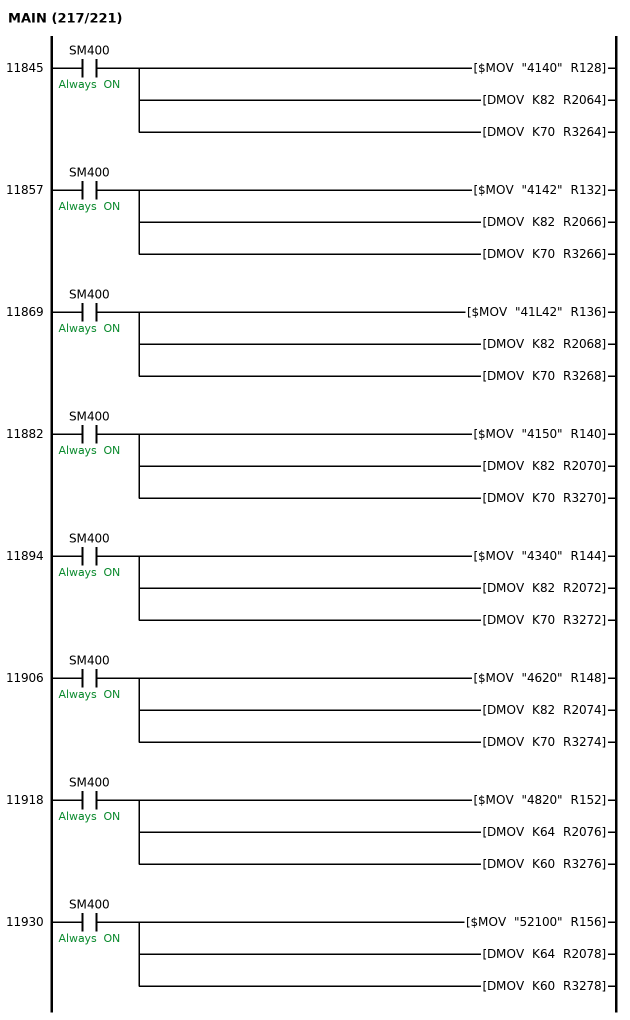
[picture p216: ladder of MAIN, rungs at steps 11845 to 11930]
11845 LD      SM400  ; Always  ON
      $MOV    "4140" R128
      DMOV    K82 R2064
      DMOV    K70 R3264
11857 LD      SM400  ; Always  ON
      $MOV    "4142" R132
      DMOV    K82 R2066
      DMOV    K70 R3266
11869 LD      SM400  ; Always  ON
      $MOV    "41L42" R136
      DMOV    K82 R2068
      DMOV    K70 R3268
11882 LD      SM400  ; Always  ON
      $MOV    "4150" R140
      DMOV    K82 R2070
      DMOV    K70 R3270
11894 LD      SM400  ; Always  ON
      $MOV    "4340" R144
      DMOV    K82 R2072
      DMOV    K70 R3272
11906 LD      SM400  ; Always  ON
      $MOV    "4620" R148
      DMOV    K82 R2074
      DMOV    K70 R3274
11918 LD      SM400  ; Always  ON
      $MOV    "4820" R152
      DMOV    K64 R2076
      DMOV    K60 R3276
11930 LD      SM400  ; Always  ON
      $MOV    "52100" R156
      DMOV    K64 R2078
      DMOV    K60 R3278
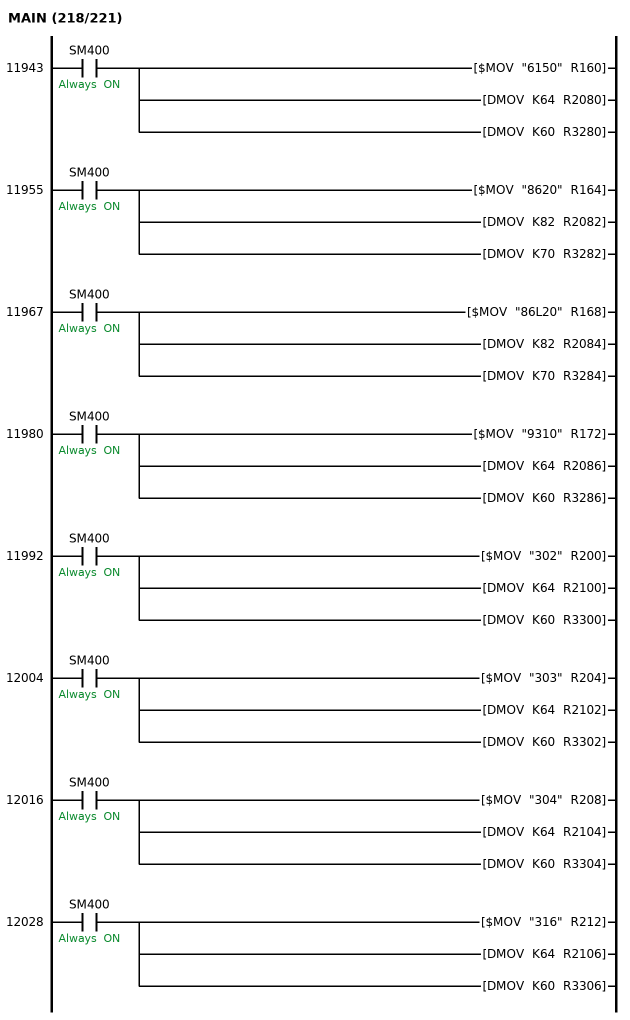
11943 LD      SM400  ; Always  ON
      $MOV    "6150" R160
      DMOV    K64 R2080
      DMOV    K60 R3280
11955 LD      SM400  ; Always  ON
      $MOV    "8620" R164
      DMOV    K82 R2082
      DMOV    K70 R3282
11967 LD      SM400  ; Always  ON
      $MOV    "86L20" R168
      DMOV    K82 R2084
      DMOV    K70 R3284
11980 LD      SM400  ; Always  ON
      $MOV    "9310" R172
      DMOV    K64 R2086
      DMOV    K60 R3286
11992 LD      SM400  ; Always  ON
      $MOV    "302" R200
      DMOV    K64 R2100
      DMOV    K60 R3300
12004 LD      SM400  ; Always  ON
      $MOV    "303" R204
      DMOV    K64 R2102
      DMOV    K60 R3302
12016 LD      SM400  ; Always  ON
      $MOV    "304" R208
      DMOV    K64 R2104
      DMOV    K60 R3304
12028 LD      SM400  ; Always  ON
      $MOV    "316" R212
      DMOV    K64 R2106
      DMOV    K60 R3306
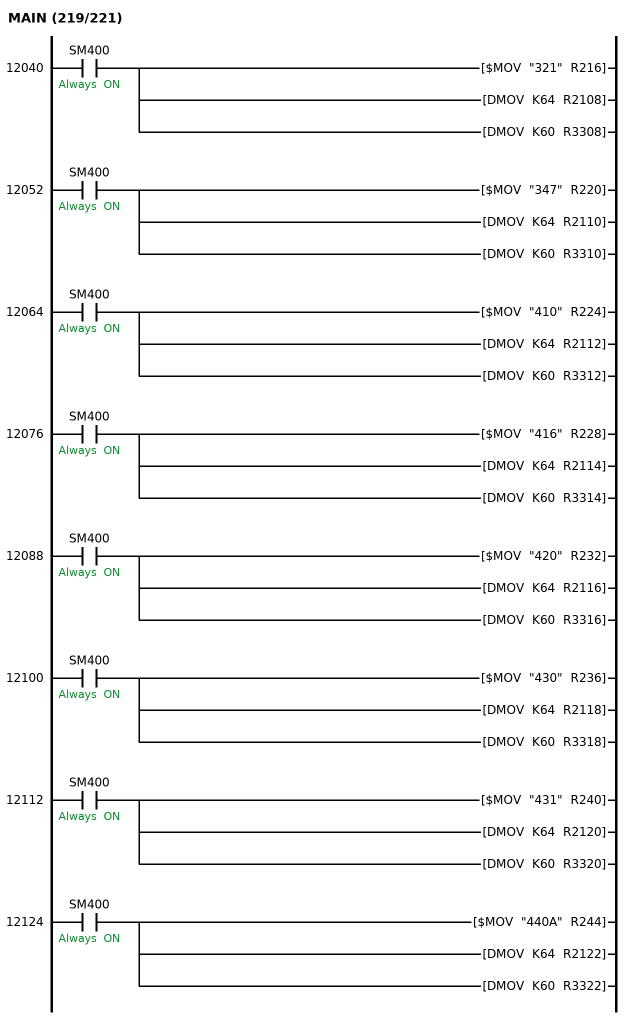
12040 LD      SM400  ; Always  ON
      $MOV    "321" R216
      DMOV    K64 R2108
      DMOV    K60 R3308
12052 LD      SM400  ; Always  ON
      $MOV    "347" R220
      DMOV    K64 R2110
      DMOV    K60 R3310
12064 LD      SM400  ; Always  ON
      $MOV    "410" R224
      DMOV    K64 R2112
      DMOV    K60 R3312
12076 LD      SM400  ; Always  ON
      $MOV    "416" R228
      DMOV    K64 R2114
      DMOV    K60 R3314
12088 LD      SM400  ; Always  ON
      $MOV    "420" R232
      DMOV    K64 R2116
      DMOV    K60 R3316
12100 LD      SM400  ; Always  ON
      $MOV    "430" R236
      DMOV    K64 R2118
      DMOV    K60 R3318
12112 LD      SM400  ; Always  ON
      $MOV    "431" R240
      DMOV    K64 R2120
      DMOV    K60 R3320
12124 LD      SM400  ; Always  ON
      $MOV    "440A" R244
      DMOV    K64 R2122
      DMOV    K60 R3322
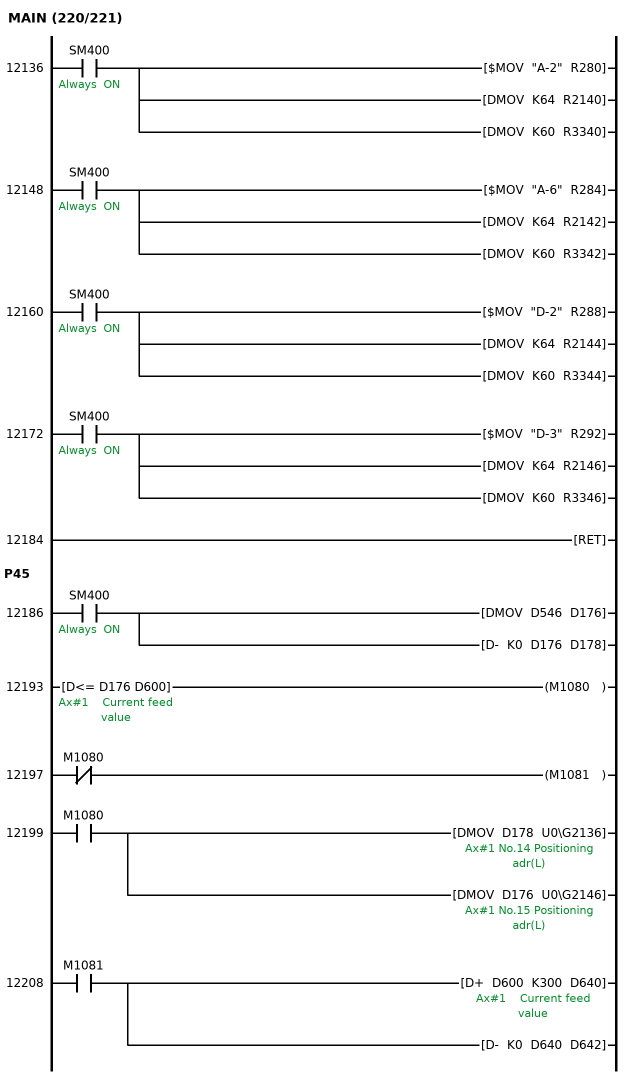
12136 LD      SM400  ; Always  ON
      $MOV    "A-2" R280
      DMOV    K64 R2140
      DMOV    K60 R3340
12148 LD      SM400  ; Always  ON
      $MOV    "A-6" R284
      DMOV    K64 R2142
      DMOV    K60 R3342
12160 LD      SM400  ; Always  ON
      $MOV    "D-2" R288
      DMOV    K64 R2144
      DMOV    K60 R3344
12172 LD      SM400  ; Always  ON
      $MOV    "D-3" R292
      DMOV    K64 R2146
      DMOV    K60 R3346
12184 RET
      P45
12186 LD      SM400  ; Always  ON
      DMOV    D546 D176
      D-      K0 D176 D178
12193 LDD<=   D176 D600  ; Ax#1    Current feed    value
      OUT     M1080
12197 LDI     M1080
      OUT     M1081
12199 LD      M1080
      DMOV    D178 U0\G2136  ; Ax#1 No.14 Positioning adr(L)
      DMOV    D176 U0\G2146  ; Ax#1 No.15 Positioning adr(L)
12208 LD      M1081
      D+      D600 K300 D640
      D-      K0 D640 D642
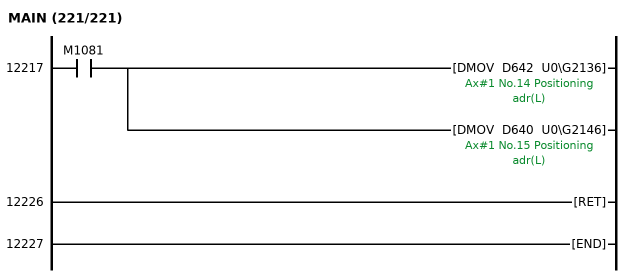
12217 LD      M1081
      DMOV    D642 U0\G2136
      DMOV    D640 U0\G2146
12226 RET
12227 END
END_PROGRAM

PROGRAM HMS
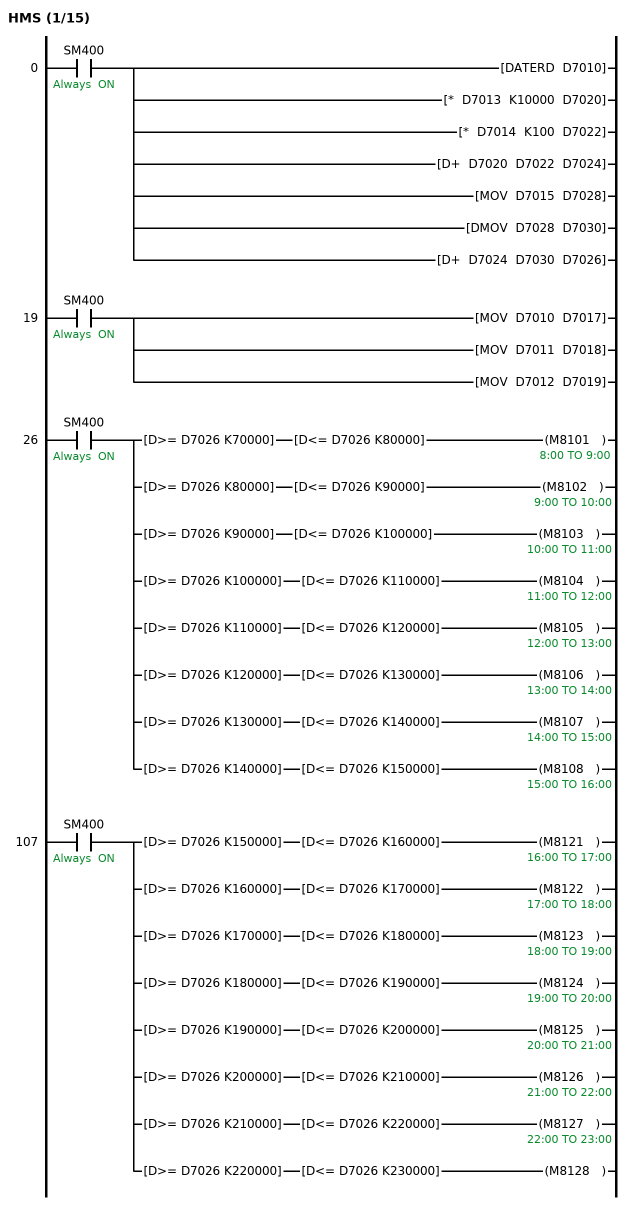
0     LD      SM400  ; Always  ON
      DATERD  D7010
      *       D7013 K10000 D7020
      *       D7014 K100 D7022
      D+      D7020 D7022 D7024
      MOV     D7015 D7028
      DMOV    D7028 D7030
      D+      D7024 D7030 D7026
19    LD      SM400  ; Always  ON
      MOV     D7010 D7017
      MOV     D7011 D7018
      MOV     D7012 D7019
26    LD      SM400  ; Always  ON
      MPS
      ANDD>=  D7026 K70000
      ANDD<=  D7026 K80000
      OUT     M8101  ; 8:00 TO 9:00
      MRD
      ANDD>=  D7026 K80000
      ANDD<=  D7026 K90000
      OUT     M8102  ; 9:00 TO 10:00
      MRD
      ANDD>=  D7026 K90000
      ANDD<=  D7026 K100000
      OUT     M8103  ; 10:00 TO 11:00
      MRD
      ANDD>=  D7026 K100000
      ANDD<=  D7026 K110000
      OUT     M8104  ; 11:00 TO 12:00
      MRD
      ANDD>=  D7026 K110000
      ANDD<=  D7026 K120000
      OUT     M8105  ; 12:00 TO 13:00
      MRD
      ANDD>=  D7026 K120000
      ANDD<=  D7026 K130000
      OUT     M8106  ; 13:00 TO 14:00
      MRD
      ANDD>=  D7026 K130000
      ANDD<=  D7026 K140000
      OUT     M8107  ; 14:00 TO 15:00
      MPP
      ANDD>=  D7026 K140000
      ANDD<=  D7026 K150000
      OUT     M8108  ; 15:00 TO 16:00
107   LD      SM400  ; Always  ON
      MPS
      ANDD>=  D7026 K150000
      ANDD<=  D7026 K160000
      OUT     M8121  ; 16:00 TO 17:00
      MRD
      ANDD>=  D7026 K160000
      ANDD<=  D7026 K170000
      OUT     M8122  ; 17:00 TO 18:00
      MRD
      ANDD>=  D7026 K170000
      ANDD<=  D7026 K180000
      OUT     M8123  ; 18:00 TO 19:00
      MRD
      ANDD>=  D7026 K180000
      ANDD<=  D7026 K190000
      OUT     M8124  ; 19:00 TO 20:00
      MRD
      ANDD>=  D7026 K190000
      ANDD<=  D7026 K200000
      OUT     M8125  ; 20:00 TO 21:00
      MRD
      ANDD>=  D7026 K200000
      ANDD<=  D7026 K210000
      OUT     M8126  ; 21:00 TO 22:00
      MRD
      ANDD>=  D7026 K210000
      ANDD<=  D7026 K220000
      OUT     M8127  ; 22:00 TO 23:00
      MPP
      ANDD>=  D7026 K220000
      ANDD<=  D7026 K230000
      OUT     M8128
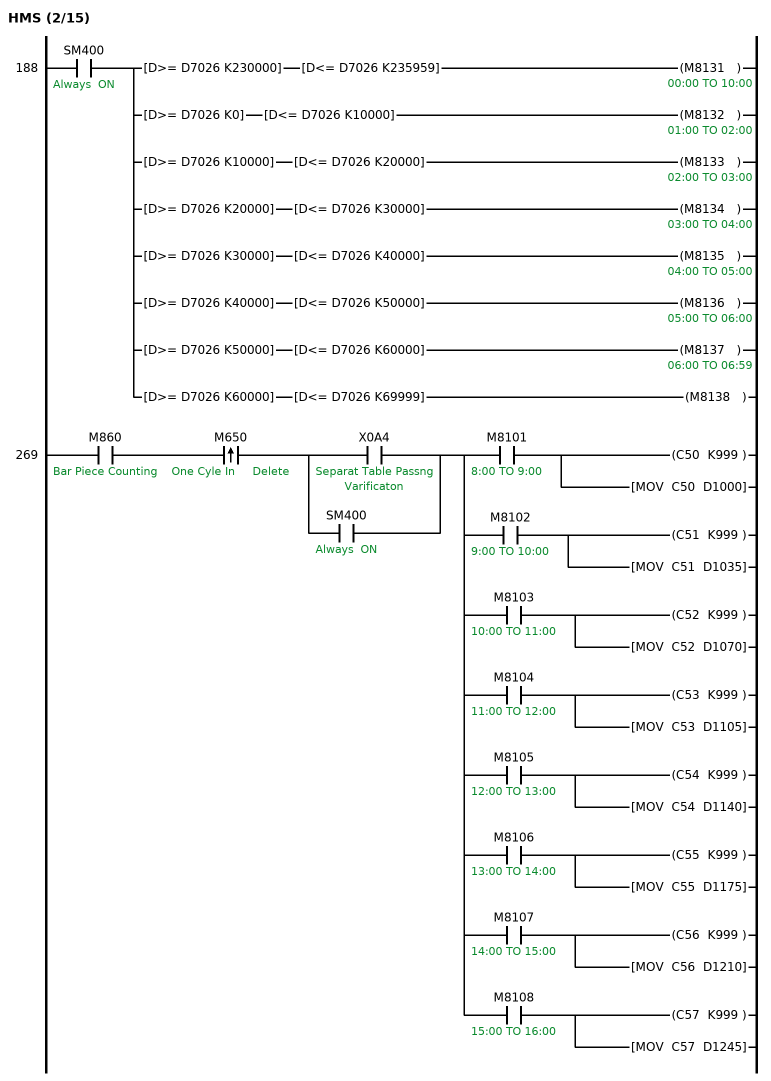
188   LD      SM400  ; Always  ON
      MPS
      ANDD>=  D7026 K230000
      ANDD<=  D7026 K235959
      OUT     M8131  ; 00:00 TO 10:00
      MRD
      ANDD>=  D7026 K0
      ANDD<=  D7026 K10000
      OUT     M8132  ; 01:00 TO 02:00
      MRD
      ANDD>=  D7026 K10000
      ANDD<=  D7026 K20000
      OUT     M8133  ; 02:00 TO 03:00
      MRD
      ANDD>=  D7026 K20000
      ANDD<=  D7026 K30000
      OUT     M8134  ; 03:00 TO 04:00
      MRD
      ANDD>=  D7026 K30000
      ANDD<=  D7026 K40000
      OUT     M8135  ; 04:00 TO 05:00
      MRD
      ANDD>=  D7026 K40000
      ANDD<=  D7026 K50000
      OUT     M8136  ; 05:00 TO 06:00
      MRD
      ANDD>=  D7026 K50000
      ANDD<=  D7026 K60000
      OUT     M8137  ; 06:00 TO 06:59
      MPP
      ANDD>=  D7026 K60000
      ANDD<=  D7026 K69999
      OUT     M8138
269   LD      M860  ; Bar Piece Counting
      ANDP    M650  ; One Cyle In     Delete
      LD      X0A4  ; Separat Table Passng Varificaton
      OR      SM400  ; Always  ON
      ANB
      MPS
      AND     M8101  ; 8:00 TO 9:00
      OUT     C50 K999
      MOV     C50 D1000
      MRD
      AND     M8102  ; 9:00 TO 10:00
      OUT     C51 K999
      MOV     C51 D1035
      MRD
      AND     M8103  ; 10:00 TO 11:00
      OUT     C52 K999
      MOV     C52 D1070
      MRD
      AND     M8104  ; 11:00 TO 12:00
      OUT     C53 K999
      MOV     C53 D1105
      MRD
      AND     M8105  ; 12:00 TO 13:00
      OUT     C54 K999
      MOV     C54 D1140
      MRD
      AND     M8106  ; 13:00 TO 14:00
      OUT     C55 K999
      MOV     C55 D1175
      MRD
      AND     M8107  ; 14:00 TO 15:00
      OUT     C56 K999
      MOV     C56 D1210
      MPP
      AND     M8108  ; 15:00 TO 16:00
      OUT     C57 K999
      MOV     C57 D1245
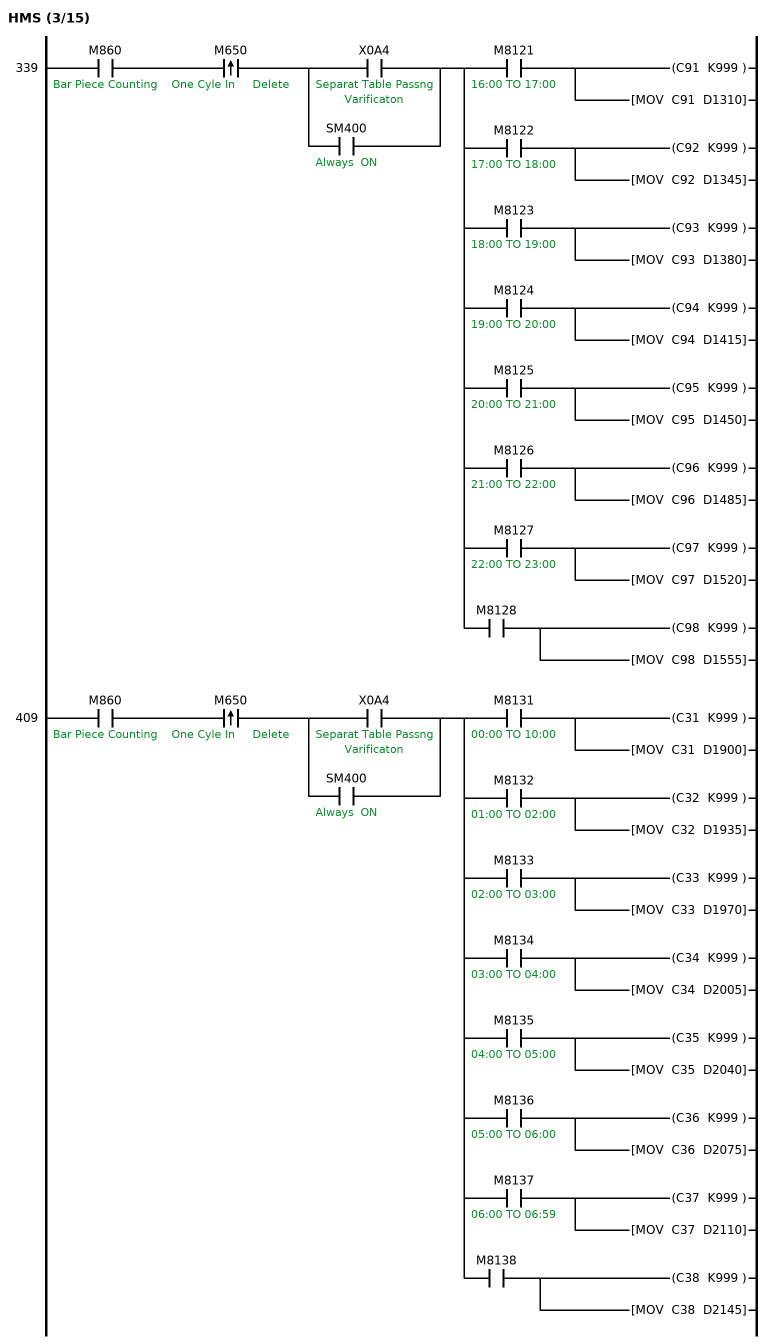
339   LD      M860  ; Bar Piece Counting
      ANDP    M650  ; One Cyle In     Delete
      LD      X0A4  ; Separat Table Passng Varificaton
      OR      SM400  ; Always  ON
      ANB
      MPS
      AND     M8121  ; 16:00 TO 17:00
      OUT     C91 K999
      MOV     C91 D1310
      MRD
      AND     M8122  ; 17:00 TO 18:00
      OUT     C92 K999
      MOV     C92 D1345
      MRD
      AND     M8123  ; 18:00 TO 19:00
      OUT     C93 K999
      MOV     C93 D1380
      MRD
      AND     M8124  ; 19:00 TO 20:00
      OUT     C94 K999
      MOV     C94 D1415
      MRD
      AND     M8125  ; 20:00 TO 21:00
      OUT     C95 K999
      MOV     C95 D1450
      MRD
      AND     M8126  ; 21:00 TO 22:00
      OUT     C96 K999
      MOV     C96 D1485
      MRD
      AND     M8127  ; 22:00 TO 23:00
      OUT     C97 K999
      MOV     C97 D1520
      MPP
      AND     M8128
      OUT     C98 K999
      MOV     C98 D1555
409   LD      M860  ; Bar Piece Counting
      ANDP    M650  ; One Cyle In     Delete
      LD      X0A4  ; Separat Table Passng Varificaton
      OR      SM400  ; Always  ON
      ANB
      MPS
      AND     M8131  ; 00:00 TO 10:00
      OUT     C31 K999
      MOV     C31 D1900
      MRD
      AND     M8132  ; 01:00 TO 02:00
      OUT     C32 K999
      MOV     C32 D1935
      MRD
      AND     M8133  ; 02:00 TO 03:00
      OUT     C33 K999
      MOV     C33 D1970
      MRD
      AND     M8134  ; 03:00 TO 04:00
      OUT     C34 K999
      MOV     C34 D2005
      MRD
      AND     M8135  ; 04:00 TO 05:00
      OUT     C35 K999
      MOV     C35 D2040
      MRD
      AND     M8136  ; 05:00 TO 06:00
      OUT     C36 K999
      MOV     C36 D2075
      MRD
      AND     M8137  ; 06:00 TO 06:59
      OUT     C37 K999
      MOV     C37 D2110
      MPP
      AND     M8138
      OUT     C38 K999
      MOV     C38 D2145
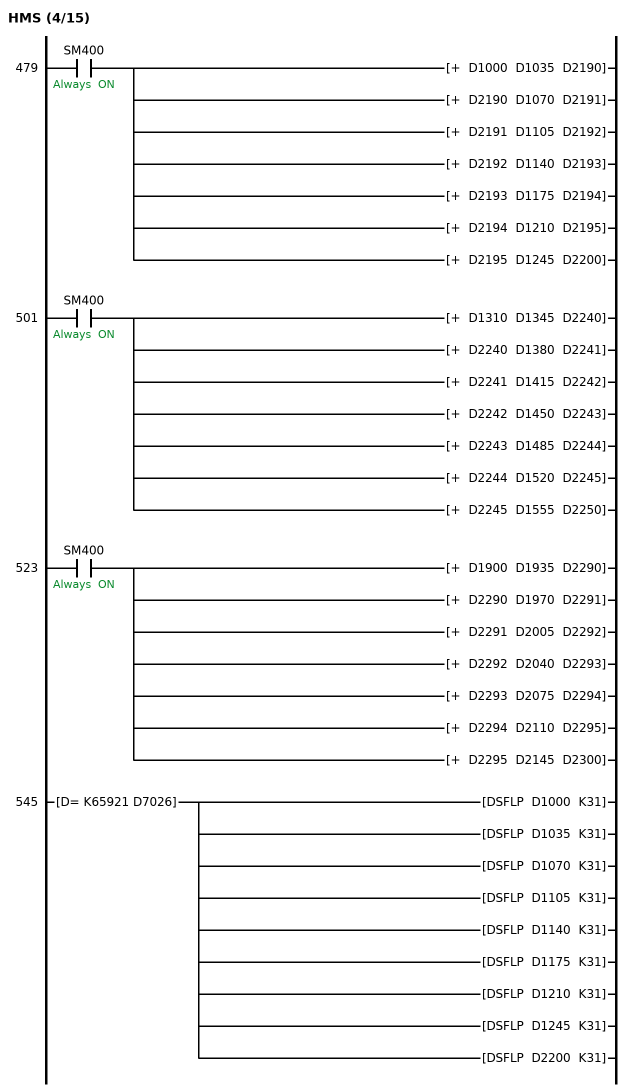
479   LD      SM400  ; Always  ON
      +       D1000 D1035 D2190
      +       D2190 D1070 D2191
      +       D2191 D1105 D2192
      +       D2192 D1140 D2193
      +       D2193 D1175 D2194
      +       D2194 D1210 D2195
      +       D2195 D1245 D2200
501   LD      SM400  ; Always  ON
      +       D1310 D1345 D2240
      +       D2240 D1380 D2241
      +       D2241 D1415 D2242
      +       D2242 D1450 D2243
      +       D2243 D1485 D2244
      +       D2244 D1520 D2245
      +       D2245 D1555 D2250
523   LD      SM400  ; Always  ON
      +       D1900 D1935 D2290
      +       D2290 D1970 D2291
      +       D2291 D2005 D2292
      +       D2292 D2040 D2293
      +       D2293 D2075 D2294
      +       D2294 D2110 D2295
      +       D2295 D2145 D2300
545   LDD=    K65921 D7026
      DSFLP   D1000 K31
      DSFLP   D1035 K31
      DSFLP   D1070 K31
      DSFLP   D1105 K31
      DSFLP   D1140 K31
      DSFLP   D1175 K31
      DSFLP   D1210 K31
      DSFLP   D1245 K31
      DSFLP   D2200 K31
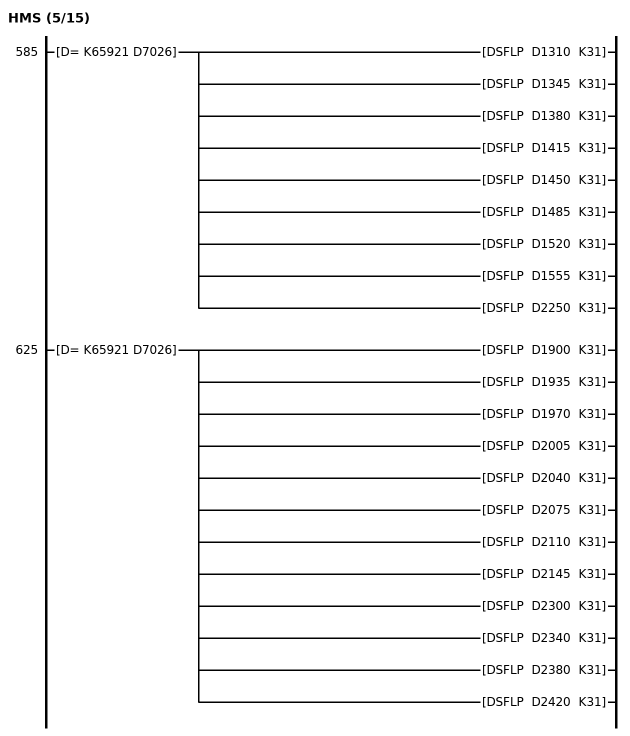
585   LDD=    K65921 D7026
      DSFLP   D1310 K31
      DSFLP   D1345 K31
      DSFLP   D1380 K31
      DSFLP   D1415 K31
      DSFLP   D1450 K31
      DSFLP   D1485 K31
      DSFLP   D1520 K31
      DSFLP   D1555 K31
      DSFLP   D2250 K31
625   LDD=    K65921 D7026
      DSFLP   D1900 K31
      DSFLP   D1935 K31
      DSFLP   D1970 K31
      DSFLP   D2005 K31
      DSFLP   D2040 K31
      DSFLP   D2075 K31
      DSFLP   D2110 K31
      DSFLP   D2145 K31
      DSFLP   D2300 K31
      DSFLP   D2340 K31
      DSFLP   D2380 K31
      DSFLP   D2420 K31
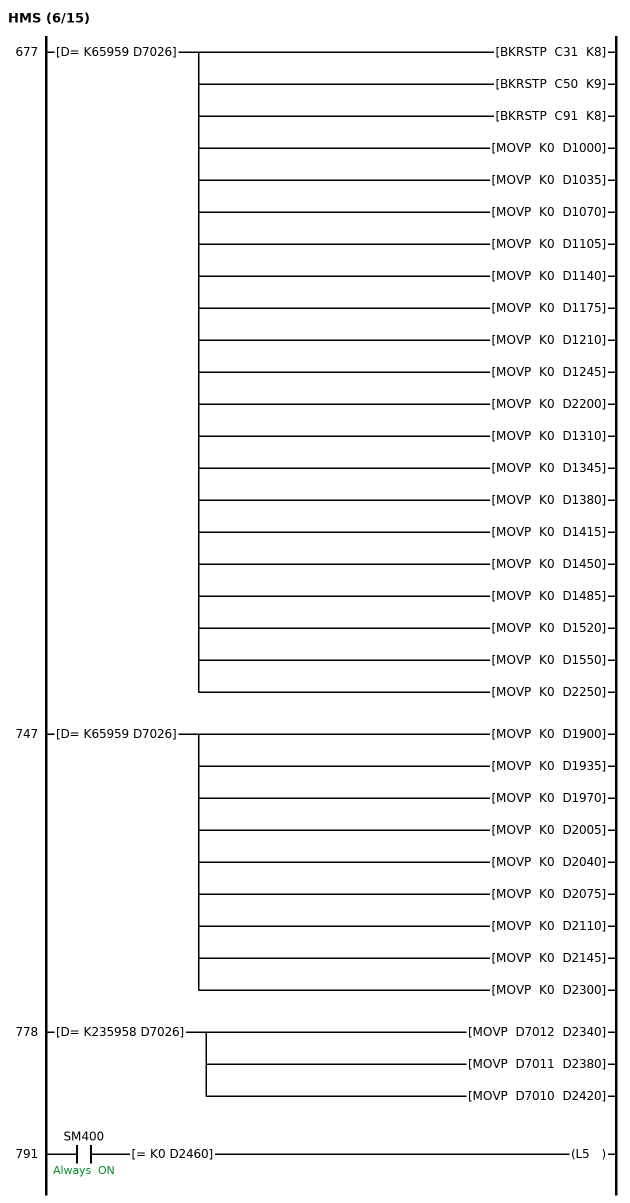
677   LDD=    K65959 D7026
      BKRSTP  C31 K8
      BKRSTP  C50 K9
      BKRSTP  C91 K8
      MOVP    K0 D1000
      MOVP    K0 D1035
      MOVP    K0 D1070
      MOVP    K0 D1105
      MOVP    K0 D1140
      MOVP    K0 D1175
      MOVP    K0 D1210
      MOVP    K0 D1245
      MOVP    K0 D2200
      MOVP    K0 D1310
      MOVP    K0 D1345
      MOVP    K0 D1380
      MOVP    K0 D1415
      MOVP    K0 D1450
      MOVP    K0 D1485
      MOVP    K0 D1520
      MOVP    K0 D1550
      MOVP    K0 D2250
747   LDD=    K65959 D7026
      MOVP    K0 D1900
      MOVP    K0 D1935
      MOVP    K0 D1970
      MOVP    K0 D2005
      MOVP    K0 D2040
      MOVP    K0 D2075
      MOVP    K0 D2110
      MOVP    K0 D2145
      MOVP    K0 D2300
778   LDD=    K235958 D7026
      MOVP    D7012 D2340
      MOVP    D7011 D2380
      MOVP    D7010 D2420
791   LD      SM400  ; Always  ON
      AND=    K0 D2460
      OUT     L5
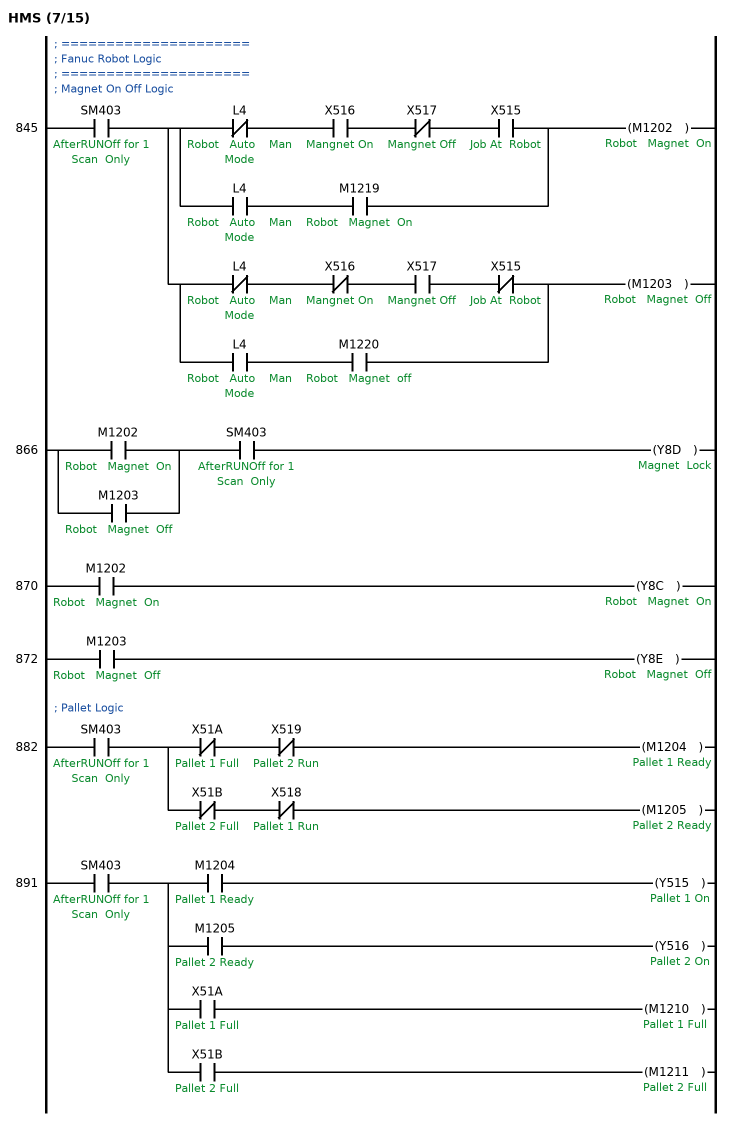
; =====================
; Fanuc Robot Logic
; =====================
; Magnet On Off Logic
845   LD      SM403  ; AfterRUNOff for 1 Scan  Only
      MPS
      LDI     L4  ; Robot   Auto    Man     Mode
      AND     X516  ; Mangnet On
      ANI     X517  ; Mangnet Off
      AND     X515  ; Job At  Robot
      LD      L4  ; Robot   Auto    Man     Mode
      AND     M1219  ; Robot   Magnet  On
      ORB
      ANB
      OUT     M1202  ; Robot   Magnet  On
      MPP
      LDI     L4  ; Robot   Auto    Man     Mode
      ANI     X516  ; Mangnet On
      AND     X517  ; Mangnet Off
      ANI     X515  ; Job At  Robot
      LD      L4  ; Robot   Auto    Man     Mode
      AND     M1220  ; Robot   Magnet  off
      ORB
      ANB
      OUT     M1203  ; Robot   Magnet  Off
866   LD      M1202  ; Robot   Magnet  On
      OR      M1203  ; Robot   Magnet  Off
      AND     SM403  ; AfterRUNOff for 1 Scan  Only
      OUT     Y8D  ; Magnet  Lock
870   LD      M1202  ; Robot   Magnet  On
      OUT     Y8C  ; Robot   Magnet  On
872   LD      M1203  ; Robot   Magnet  Off
      OUT     Y8E  ; Robot   Magnet  Off
; Pallet Logic
882   LD      SM403  ; AfterRUNOff for 1 Scan  Only
      MPS
      ANI     X51A  ; Pallet 1 Full
      ANI     X519  ; Pallet 2 Run
      OUT     M1204  ; Pallet 1 Ready
      MPP
      ANI     X51B  ; Pallet 2 Full
      ANI     X518  ; Pallet 1 Run
      OUT     M1205  ; Pallet 2 Ready
891   LD      SM403  ; AfterRUNOff for 1 Scan  Only
      MPS
      AND     M1204  ; Pallet 1 Ready
      OUT     Y515  ; Pallet 1 On
      MRD
      AND     M1205  ; Pallet 2 Ready
      OUT     Y516  ; Pallet 2 On
      MRD
      AND     X51A  ; Pallet 1 Full
      OUT     M1210  ; Pallet 1 Full
      MPP
      AND     X51B  ; Pallet 2 Full
      OUT     M1211  ; Pallet 2 Full
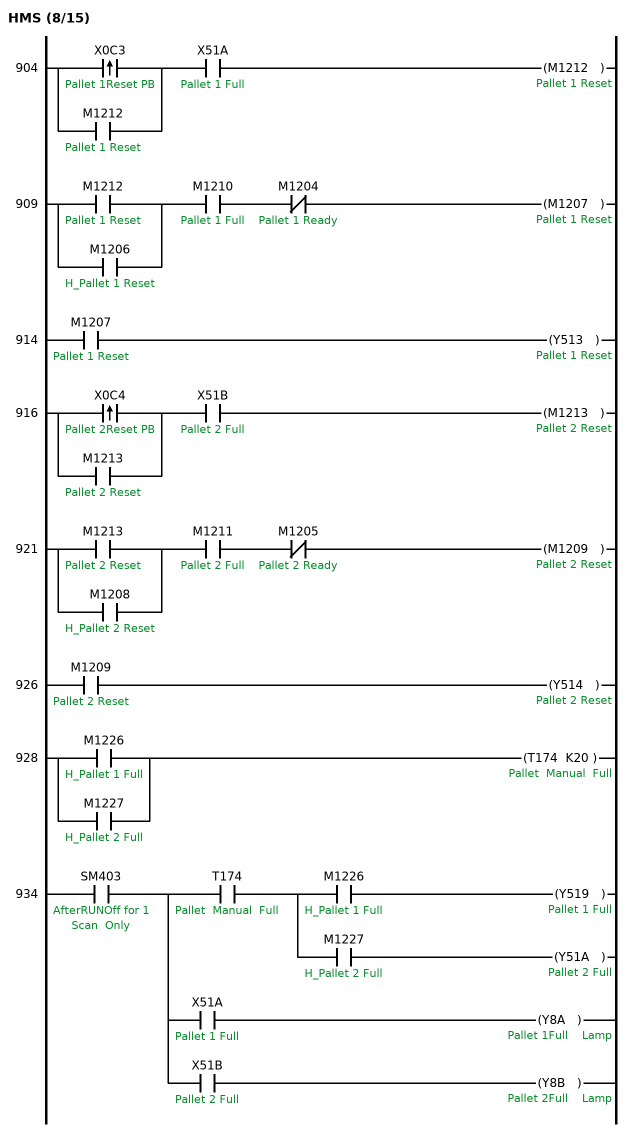
904   LDP     X0C3  ; Pallet 1Reset PB
      OR      M1212  ; Pallet 1 Reset
      AND     X51A  ; Pallet 1 Full
      OUT     M1212  ; Pallet 1 Reset
909   LD      M1212  ; Pallet 1 Reset
      OR      M1206  ; H_Pallet 1 Reset
      AND     M1210  ; Pallet 1 Full
      ANI     M1204  ; Pallet 1 Ready
      OUT     M1207  ; Pallet 1 Reset
914   LD      M1207  ; Pallet 1 Reset
      OUT     Y513  ; Pallet 1 Reset
916   LDP     X0C4  ; Pallet 2Reset PB
      OR      M1213  ; Pallet 2 Reset
      AND     X51B  ; Pallet 2 Full
      OUT     M1213  ; Pallet 2 Reset
921   LD      M1213  ; Pallet 2 Reset
      OR      M1208  ; H_Pallet 2 Reset
      AND     M1211  ; Pallet 2 Full
      ANI     M1205  ; Pallet 2 Ready
      OUT     M1209  ; Pallet 2 Reset
926   LD      M1209  ; Pallet 2 Reset
      OUT     Y514  ; Pallet 2 Reset
928   LD      M1226  ; H_Pallet 1 Full
      OR      M1227  ; H_Pallet 2 Full
      OUT     T174 K20  ; Pallet  Manual  Full
934   LD      SM403  ; AfterRUNOff for 1 Scan  Only
      MPS
      AND     T174  ; Pallet  Manual  Full
      MPS
      AND     M1226  ; H_Pallet 1 Full
      OUT     Y519  ; Pallet 1 Full
      MPP
      AND     M1227  ; H_Pallet 2 Full
      OUT     Y51A  ; Pallet 2 Full
      MRD
      AND     X51A  ; Pallet 1 Full
      OUT     Y8A  ; Pallet 1Full    Lamp
      MPP
      AND     X51B  ; Pallet 2 Full
      OUT     Y8B  ; Pallet 2Full    Lamp
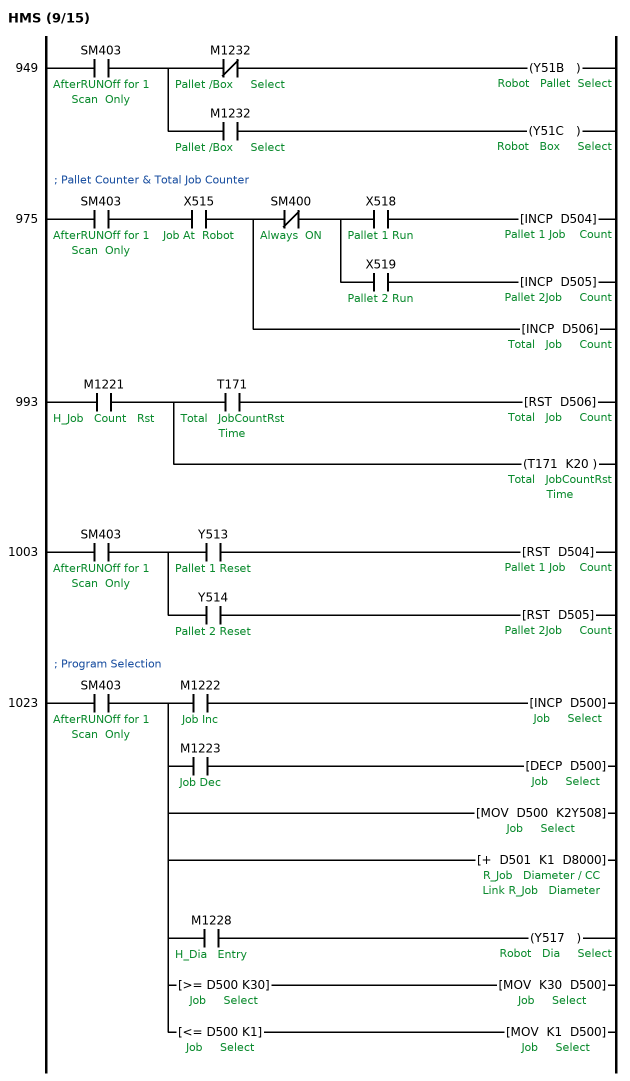
949   LD      SM403  ; AfterRUNOff for 1 Scan  Only
      MPS
      ANI     M1232  ; Pallet /Box     Select
      OUT     Y51B  ; Robot   Pallet  Select
      MPP
      AND     M1232  ; Pallet /Box     Select
      OUT     Y51C  ; Robot   Box     Select
; Pallet Counter & Total Job Counter
975   LD      SM403  ; AfterRUNOff for 1 Scan  Only
      AND     X515  ; Job At  Robot
      MPS
      ANI     SM400  ; Always  ON
      MPS
      AND     X518  ; Pallet 1 Run
      INCP    D504  ; Pallet 1 Job    Count
      MPP
      AND     X519  ; Pallet 2 Run
      INCP    D505  ; Pallet 2Job     Count
      MPP
      INCP    D506  ; Total   Job     Count
993   LD      M1221  ; H_Job   Count   Rst
      MPS
      AND     T171  ; Total   JobCountRst Time
      RST     D506  ; Total   Job     Count
      MPP
      OUT     T171 K20  ; Total   JobCountRst Time
1003  LD      SM403  ; AfterRUNOff for 1 Scan  Only
      MPS
      AND     Y513  ; Pallet 1 Reset
      RST     D504  ; Pallet 1 Job    Count
      MPP
      AND     Y514  ; Pallet 2 Reset
      RST     D505  ; Pallet 2Job     Count
; Program Selection
1023  LD      SM403  ; AfterRUNOff for 1 Scan  Only
      MPS
      AND     M1222  ; Job Inc
      INCP    D500  ; Job     Select
      MRD
      AND     M1223  ; Job Dec
      DECP    D500
      MPP
      MOV     D500 K2Y508  ; PNS 1   Style 1
      +       D501 K1 D8000  ; R_Job   Diameter / CC Link R_Job   Diameter
      MPS
      AND     M1228  ; H_Dia   Entry
      OUT     Y517  ; Robot   Dia     Select
      MRD
      AND>=   D500 K30  ; Job     Select
      MOV     K30 D500
      MPP
      AND<=   D500 K1  ; Job     Select
      MOV     K1 D500
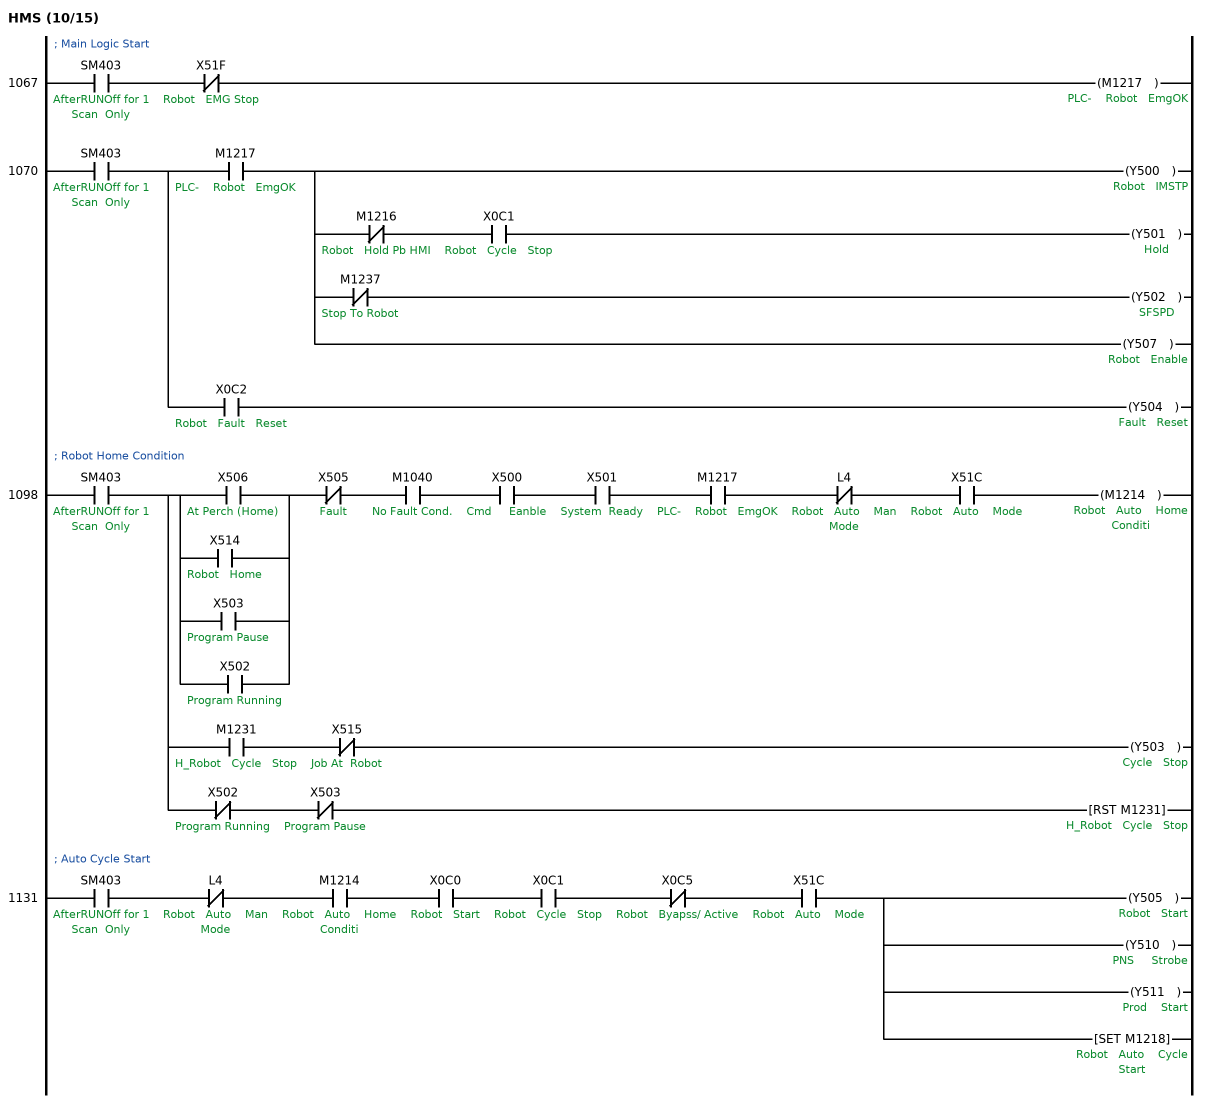
; Main Logic Start
1067  LD      SM403  ; AfterRUNOff for 1 Scan  Only
      ANI     X51F  ; Robot   EMG Stop
      OUT     M1217  ; PLC-    Robot   EmgOK
1070  LD      SM403  ; AfterRUNOff for 1 Scan  Only
      MPS
      AND     M1217  ; PLC-    Robot   EmgOK
      OUT     Y500  ; Robot   IMSTP
      MPS
      ANI     M1216  ; Robot   Hold Pb HMI
      AND     X0C1  ; Robot   Cycle   Stop
      OUT     Y501  ; Hold
      MRD
      ANI     M1237  ; Stop To Robot
      OUT     Y502  ; SFSPD
      MPP
      OUT     Y507  ; Robot   Enable
      MPP
      AND     X0C2  ; Robot   Fault   Reset
      OUT     Y504  ; Fault   Reset
; Robot Home Condition
1098  LD      SM403  ; AfterRUNOff for 1 Scan  Only
      MPS
      LD      X506  ; At Perch (Home)
      OR      X514  ; Robot   Home
      OR      X503  ; Program Pause
      OR      X502  ; Program Running
      ANB
      ANI     X505  ; Fault
      AND     M1040  ; No Fault Cond.
      AND     X500  ; Cmd     Eanble
      AND     X501  ; System  Ready
      AND     M1217  ; PLC-    Robot   EmgOK
      ANI     L4  ; Robot   Auto    Man     Mode
      AND     X51C  ; Robot   Auto    Mode
      OUT     M1214  ; Robot   Auto    Home    Conditi
      MRD
      AND     M1231  ; H_Robot   Cycle   Stop
      ANI     X515  ; Job At  Robot
      OUT     Y503  ; Cycle   Stop
      MPP
      ANI     X502  ; Program Running
      ANI     X503  ; Program Pause
      RST     M1231  ; H_Robot   Cycle   Stop
; Auto Cycle Start
1131  LD      SM403  ; AfterRUNOff for 1 Scan  Only
      ANI     L4  ; Robot   Auto    Man     Mode
      AND     M1214  ; Robot   Auto    Home    Conditi
      AND     X0C0  ; Robot   Start
      AND     X0C1  ; Robot   Cycle   Stop
      ANI     X0C5  ; Robot   Byapss/ Active
      AND     X51C  ; Robot   Auto    Mode
      OUT     Y505  ; Robot   Start
      OUT     Y510  ; PNS     Strobe
      OUT     Y511  ; Prod    Start
      SET     M1218  ; Robot   Auto    Cycle   Start
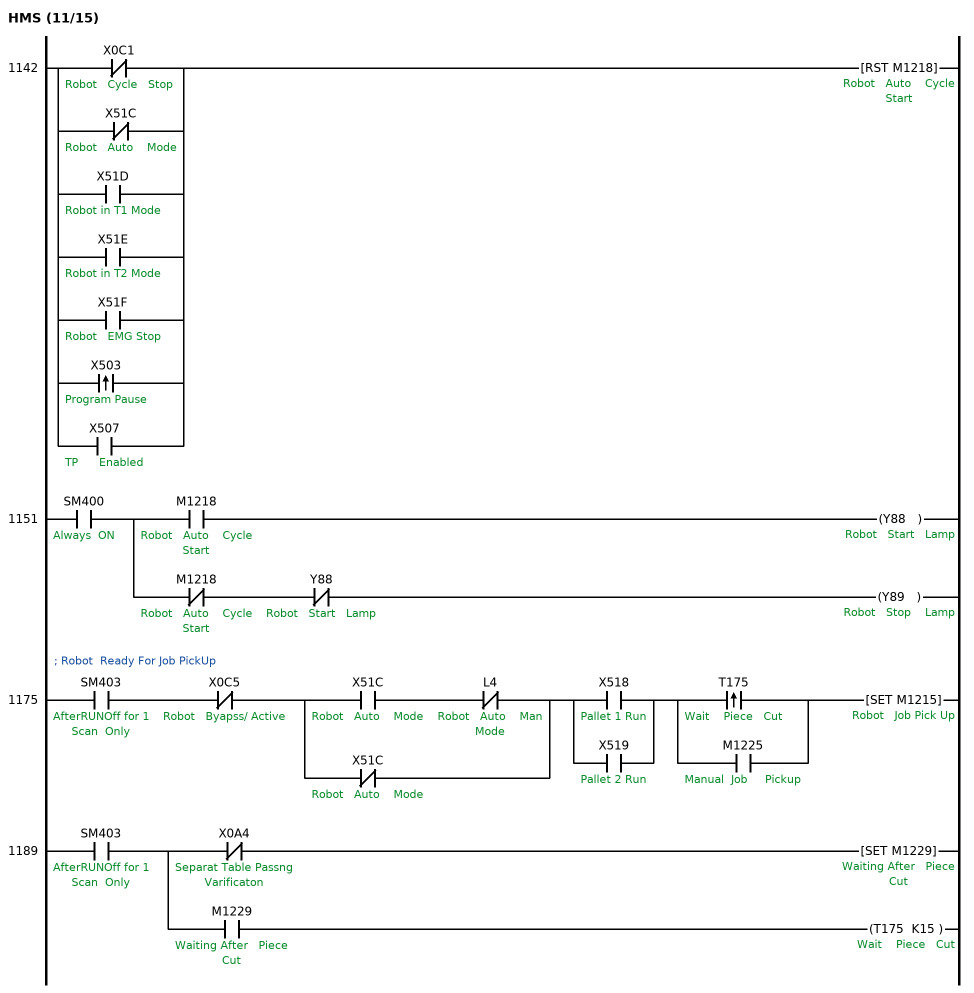
1142  LDI     X0C1  ; Robot   Cycle   Stop
      ORI     X51C  ; Robot   Auto    Mode
      OR      X51D  ; Robot in T1 Mode
      OR      X51E  ; Robot in T2 Mode
      OR      X51F  ; Robot   EMG Stop
      ORP     X503  ; Program Pause
      OR      X507  ; TP      Enabled
      RST     M1218  ; Robot   Auto    Cycle   Start
1151  LD      SM400  ; Always  ON
      MPS
      AND     M1218  ; Robot   Auto    Cycle   Start
      OUT     Y88  ; Robot   Start   Lamp
      MPP
      ANI     M1218  ; Robot   Auto    Cycle   Start
      ANI     Y88  ; Robot   Start   Lamp
      OUT     Y89  ; Robot   Stop    Lamp
; Robot  Ready For Job PickUp
1175  LD      SM403  ; AfterRUNOff for 1 Scan  Only
      ANI     X0C5  ; Robot   Byapss/ Active
      LD      X51C  ; Robot   Auto    Mode
      ANI     L4  ; Robot   Auto    Man     Mode
      ORI     X51C  ; Robot   Auto    Mode
      ANB
      LD      X518  ; Pallet 1 Run
      OR      X519  ; Pallet 2 Run
      ANB
      LDP     T175  ; Wait    Piece   Cut
      OR      M1225  ; Manual  Job     Pickup
      ANB
      SET     M1215  ; Robot   Job Pick Up
1189  LD      SM403  ; AfterRUNOff for 1 Scan  Only
      MPS
      ANI     X0A4  ; Separat Table Passng Varificaton
      SET     M1229  ; Waiting After   Piece   Cut
      MPP
      AND     M1229  ; Waiting After   Piece   Cut
      OUT     T175 K15  ; Wait    Piece   Cut
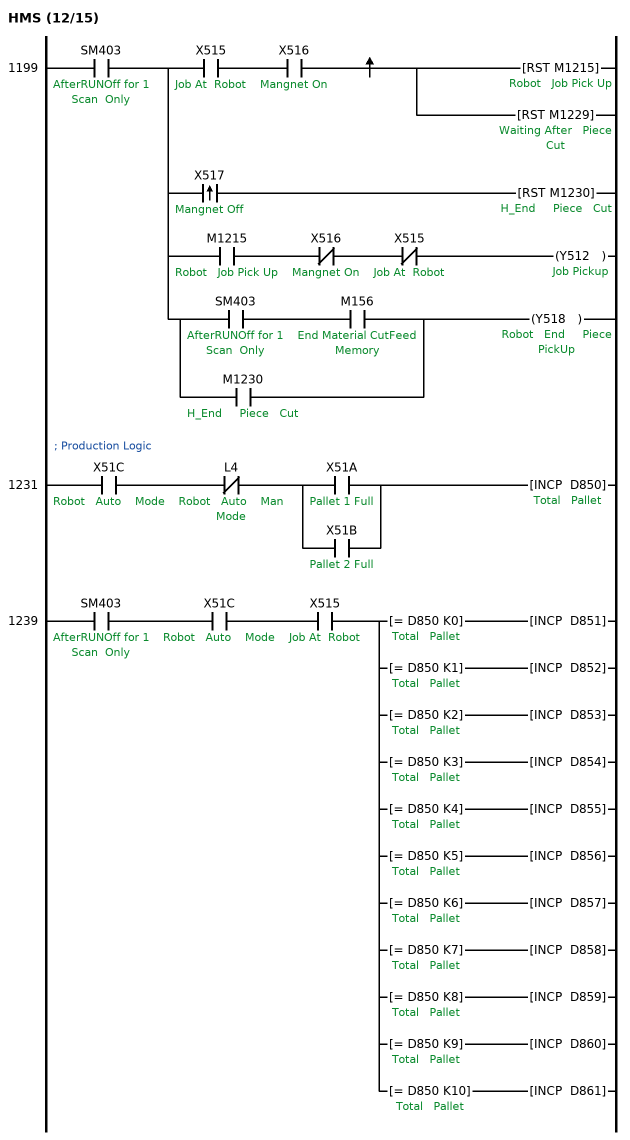
1199  LD      SM403  ; AfterRUNOff for 1 Scan  Only
      MPS
      AND     X515  ; Job At  Robot
      AND     X516  ; Mangnet On
      MEP
      RST     M1215  ; Robot   Job Pick Up
      RST     M1229  ; Waiting After   Piece   Cut
      MRD
      ANDP    X517  ; Mangnet Off
      RST     M1230  ; H_End     Piece   Cut
      MRD
      AND     M1215  ; Robot   Job Pick Up
      ANI     X516  ; Mangnet On
      ANI     X515  ; Job At  Robot
      OUT     Y512  ; Job Pickup
      MPP
      LD      SM403  ; AfterRUNOff for 1 Scan  Only
      AND     M156  ; End Material CutFeed Memory
      OR      M1230  ; H_End     Piece   Cut
      ANB
      OUT     Y518  ; Robot   End     Piece   PickUp
; Production Logic
1231  LD      X51C  ; Robot   Auto    Mode
      ANI     L4  ; Robot   Auto    Man     Mode
      LD      X51A  ; Pallet 1 Full
      OR      X51B  ; Pallet 2 Full
      ANB
      INCP    D850  ; Total   Pallet
1239  LD      SM403  ; AfterRUNOff for 1 Scan  Only
      AND     X51C  ; Robot   Auto    Mode
      AND     X515  ; Job At  Robot
      MPS
      AND=    D850 K0  ; Total   Pallet
      INCP    D851
      MRD
      AND=    D850 K1  ; Total   Pallet
      INCP    D852
      MRD
      AND=    D850 K2  ; Total   Pallet
      INCP    D853
      MRD
      AND=    D850 K3  ; Total   Pallet
      INCP    D854
      MRD
      AND=    D850 K4  ; Total   Pallet
      INCP    D855
      MRD
      AND=    D850 K5  ; Total   Pallet
      INCP    D856
      MRD
      AND=    D850 K6  ; Total   Pallet
      INCP    D857
      MRD
      AND=    D850 K7  ; Total   Pallet
      INCP    D858
      MRD
      AND=    D850 K8  ; Total   Pallet
      INCP    D859
      MRD
      AND=    D850 K9  ; Total   Pallet
      INCP    D860
      MPP
      AND=    D850 K10  ; Total   Pallet
      INCP    D861
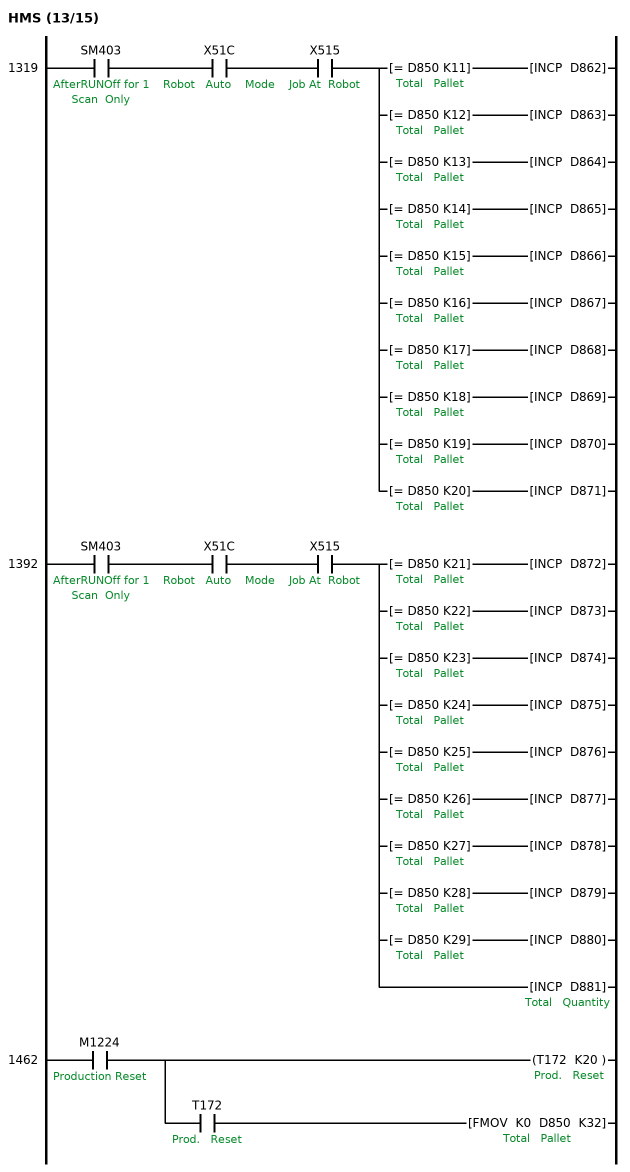
1319  LD      SM403  ; AfterRUNOff for 1 Scan  Only
      AND     X51C  ; Robot   Auto    Mode
      AND     X515  ; Job At  Robot
      MPS
      AND=    D850 K11  ; Total   Pallet
      INCP    D862
      MRD
      AND=    D850 K12  ; Total   Pallet
      INCP    D863
      MRD
      AND=    D850 K13  ; Total   Pallet
      INCP    D864
      MRD
      AND=    D850 K14  ; Total   Pallet
      INCP    D865
      MRD
      AND=    D850 K15  ; Total   Pallet
      INCP    D866
      MRD
      AND=    D850 K16  ; Total   Pallet
      INCP    D867
      MRD
      AND=    D850 K17  ; Total   Pallet
      INCP    D868
      MRD
      AND=    D850 K18  ; Total   Pallet
      INCP    D869
      MRD
      AND=    D850 K19  ; Total   Pallet
      INCP    D870
      MPP
      AND=    D850 K20  ; Total   Pallet
      INCP    D871
1392  LD      SM403  ; AfterRUNOff for 1 Scan  Only
      AND     X51C  ; Robot   Auto    Mode
      AND     X515  ; Job At  Robot
      MPS
      AND=    D850 K21  ; Total   Pallet
      INCP    D872
      MRD
      AND=    D850 K22  ; Total   Pallet
      INCP    D873
      MRD
      AND=    D850 K23  ; Total   Pallet
      INCP    D874
      MRD
      AND=    D850 K24  ; Total   Pallet
      INCP    D875
      MRD
      AND=    D850 K25  ; Total   Pallet
      INCP    D876
      MRD
      AND=    D850 K26  ; Total   Pallet
      INCP    D877
      MRD
      AND=    D850 K27  ; Total   Pallet
      INCP    D878
      MRD
      AND=    D850 K28  ; Total   Pallet
      INCP    D879
      MRD
      AND=    D850 K29  ; Total   Pallet
      INCP    D880
      MPP
      INCP    D881  ; Total   Quantity
1462  LD      M1224  ; Production Reset
      OUT     T172 K20  ; Prod.   Reset
      AND     T172  ; Prod.   Reset
      FMOV    K0 D850 K32
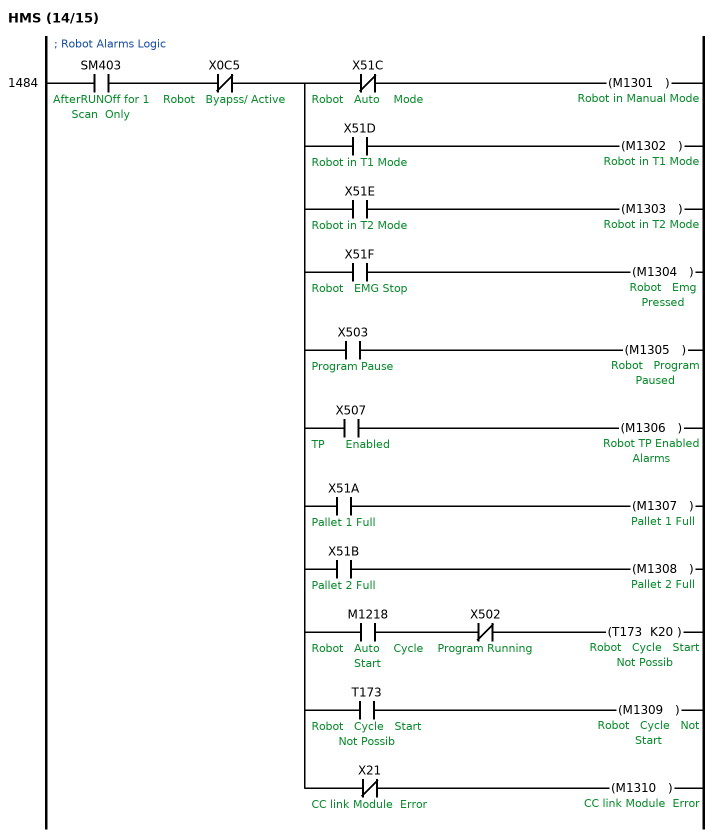
; Robot Alarms Logic
1484  LD      SM403  ; AfterRUNOff for 1 Scan  Only
      ANI     X0C5  ; Robot   Byapss/ Active
      MPS
      ANI     X51C  ; Robot   Auto    Mode
      OUT     M1301  ; Robot in Manual Mode
      MRD
      AND     X51D  ; Robot in T1 Mode
      OUT     M1302  ; Robot in T1 Mode
      MRD
      AND     X51E  ; Robot in T2 Mode
      OUT     M1303  ; Robot in T2 Mode
      MRD
      AND     X51F  ; Robot   EMG Stop
      OUT     M1304  ; Robot   Emg     Pressed
      MRD
      AND     X503  ; Program Pause
      OUT     M1305  ; Robot   Program Paused
      MRD
      AND     X507  ; TP      Enabled
      OUT     M1306  ; Robot TP Enabled Alarms
      MRD
      AND     X51A  ; Pallet 1 Full
      OUT     M1307  ; Pallet 1 Full
      MRD
      AND     X51B  ; Pallet 2 Full
      OUT     M1308  ; Pallet 2 Full
      MRD
      AND     M1218  ; Robot   Auto    Cycle   Start
      ANI     X502  ; Program Running
      OUT     T173 K20  ; Robot   Cycle   Start Not Possib
      MRD
      AND     T173  ; Robot   Cycle   Start Not Possib
      OUT     M1309  ; Robot   Cycle   Not     Start
      MPP
      ANI     X21  ; CC link Module  Error
      OUT     M1310  ; CC link Module  Error
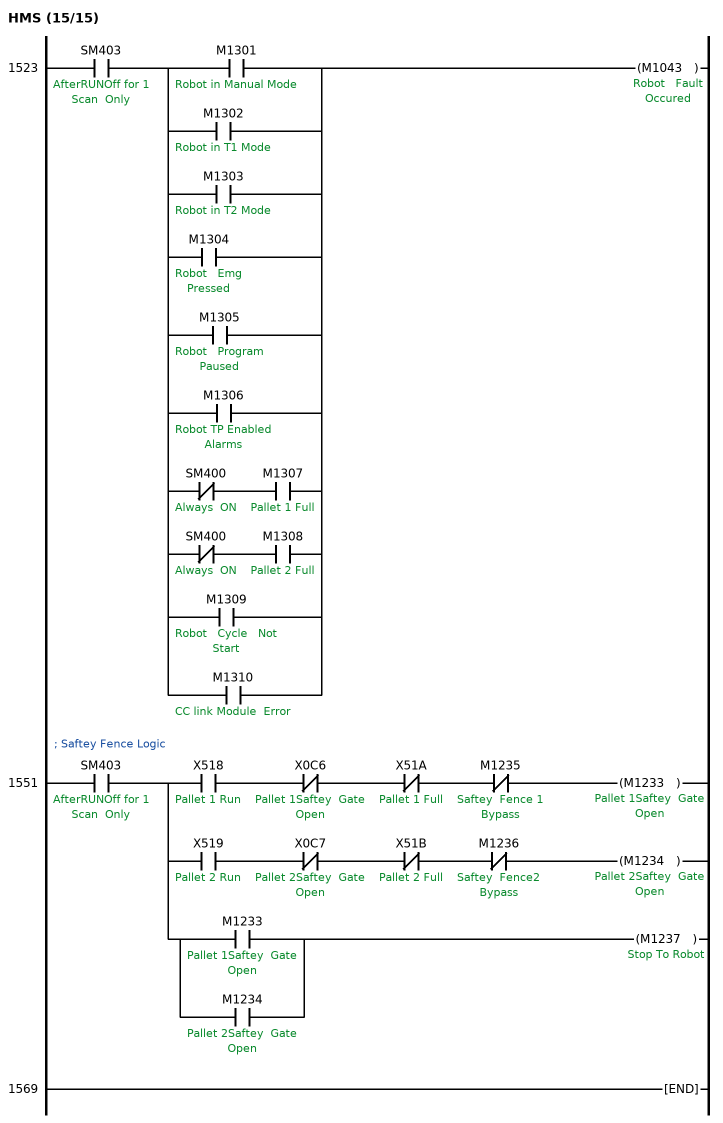
1523  LD      SM403  ; AfterRUNOff for 1 Scan  Only
      LD      M1301  ; Robot in Manual Mode
      OR      M1302  ; Robot in T1 Mode
      OR      M1303  ; Robot in T2 Mode
      OR      M1304  ; Robot   Emg     Pressed
      OR      M1305  ; Robot   Program Paused
      OR      M1306  ; Robot TP Enabled Alarms
      LDI     SM400  ; Always  ON
      AND     M1307  ; Pallet 1 Full
      ORB
      LDI     SM400  ; Always  ON
      AND     M1308  ; Pallet 2 Full
      ORB
      OR      M1309  ; Robot   Cycle   Not     Start
      OR      M1310  ; CC link Module  Error
      ANB
      OUT     M1043  ; Robot   Fault   Occured
; Saftey Fence Logic
1551  LD      SM403  ; AfterRUNOff for 1 Scan  Only
      MPS
      AND     X518  ; Pallet 1 Run
      ANI     X0C6  ; Pallet 1Saftey  Gate    Open
      ANI     X51A  ; Pallet 1 Full
      ANI     M1235  ; Saftey  Fence 1 Bypass
      OUT     M1233  ; Pallet 1Saftey  Gate    Open
      MRD
      AND     X519  ; Pallet 2 Run
      ANI     X0C7  ; Pallet 2Saftey  Gate    Open
      ANI     X51B  ; Pallet 2 Full
      ANI     M1236  ; Saftey  Fence2  Bypass
      OUT     M1234  ; Pallet 2Saftey  Gate    Open
      MPP
      LD      M1233  ; Pallet 1Saftey  Gate    Open
      OR      M1234  ; Pallet 2Saftey  Gate    Open
      ANB
      OUT     M1237  ; Stop To Robot
1569  END
END_PROGRAM

// device comments not shown above
X504  ; Motion Held
X508  ; Battery Alarms
X509  ; Busy
X50A  ; Ack 1/SN01
X50B  ; Ack 2/SN02
X50C  ; Ack 3/SN03
X50D  ; Ack 4/SN04
X50E  ; Ack 5/SN05
X50F  ; Ack 6/SN06
X510  ; Ack 7/SN07
X511  ; Ack 8/SN08
X512  ; Snack
X513  ; Reserved
B201  ; Saw Head Fwd/Bwd  Enable
B202  ; GFC Wise Clamp/Unclamp Enable
B203  ; GFC feed Fwd/Bwd Enable
B204  ; Lader Up/Dn enable
B205  ; Work Stop Fwd/Bwd Enable
B206  ; Float wise On/Off Enable
B207  ; Float work On/Off Enable
B208  ; Seperation Trim/work Enable
B20B  ; Mist ON/Off Enable
B20C  ; Air Blow On/Off Enable
B210  ; Rotary Table fwd/ bwd  Enable
B211  ; Rotary Table ON/ OFF  Enable
B212  ; Lifting Enable
D5100  ; Job ListData    Table
Y506  ; Robot Home
Y509  ; PNS 2Style 2
Y50A  ; PNS 3Style 3
Y50B  ; PNS 4Style 4
Y50C  ; PNS 5Style 5
Y50D  ; PNS 6Style 6
Y50E  ; PNS 7Style 7
Y50F  ; PNS 8Style 8
Y51D  ; Robot DI 76
Y51E  ; Robot DI 77
Y51F  ; Robot DI 78
